FUNCTION_BLOCK COUNTER (* Composite Function Block Type *)
  (* Standard: 61499-2 *)
  (* Version 0.0, 2/4/2026, SESA713705, Schneider Electric, template *)
  PACKAGE SE.Nereda;
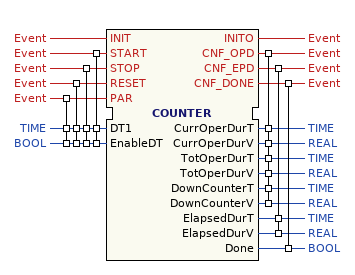
  EVENT_INPUT
    INIT;
    START WITH DT1, EnableDT; (* Begin Delay *)
    STOP WITH DT1, EnableDT; (* Cancel Delay *)
    RESET WITH DT1, EnableDT;
    PAR WITH DT1, EnableDT;
  END_EVENT
  EVENT_OUTPUT
    INITO;
    CNF_OPD WITH CurrOperDurT, CurrOperDurV, TotOperDurT, TotOperDurV, DownCounterT, DownCounterV; (* Execution Confirmation of current and total device operation duration *)
    CNF_EPD WITH ElapsedDurT, ElapsedDurV; (* Execution Confirmation of current and total Elapsed device duration *)
    CNF_DONE WITH Done;
  END_EVENT
  VAR_INPUT
    DT1 : TIME;
    EnableDT : BOOL;
  END_VAR
  VAR_OUTPUT
    CurrOperDurT : TIME;
    CurrOperDurV : REAL;
    TotOperDurT : TIME;
    TotOperDurV : REAL;
    DownCounterT : TIME;
    DownCounterV : REAL;
    ElapsedDurT : TIME;
    ElapsedDurV : REAL;
    Done : BOOL;
  END_VAR
  FBS
    IThis : COUNTER_HMI(QI := TRUE);
    CounterDurationCalc : devMntCalc(TBaseOperationDuration := T#1s, TBaseElapsedDuration := T#1d);
    CounterManager : CounterBasic;
    OPD : UDINT2TIME_2;
    REAL_OPD : UDINT2REAL_2;
    EPD_TIME : ElapsedTimeBasic;
    Counter : CounterSp;
    Smooth : boolValueChanged;
    DownCounteReal : SUB_2;
    Time2Real : TIME2REAL; {SET_ATTRIBUTE(Configuration.Component.HideUnusedPorts, )}
    Real2Time : REAL2TIME;
  END_FBS
  EVENT_CONNECTIONS
    CounterDurationCalc.INITO TO INITO;
    START TO CounterManager.DD7C28FB9184AAEE;
    STOP TO CounterManager.E0BAE2B19D215A1B;
    CounterManager.C2AFBA6527CC7C56 TO CounterDurationCalc.REQ_PV;
    Real2Time.79B40746AB555956 TO OPD.9954577AA24F9DD6;
    REAL_OPD.6FC99A5BD1C38561 TO CNF_OPD;
    EPD_TIME.B1E2A620E35E48BA TO CNF_EPD;
    OPD.79B40746AB555956 TO REAL_OPD.DD5870AA881150BB;
    REAL_OPD.6FC99A5BD1C38561 TO EPD_TIME.3E14346F747403ED;
    START TO EPD_TIME.90013566B02D29C0;
    STOP TO EPD_TIME.92EFFFA7C76F84E6;
    STOP TO EPD_TIME.3E14346F747403ED;
    Counter.C5DB08088DE67568 TO Smooth.REQ;
    PAR TO Counter.3BAEFB620E0425F5;
    REAL_OPD.6FC99A5BD1C38561 TO Counter.05FD3DED10D7909C;
    START TO Counter.C8BF0B5DBAF12ADE;
    STOP TO Counter.A678C75868BE7A7E;
    Smooth.CHD TO CNF_DONE;
    CounterDurationCalc.CNF_OPD TO Time2Real.9954577AA24F9DD6;
    PAR TO Time2Real.9954577AA24F9DD6;
    Time2Real.79B40746AB555956 TO DownCounteReal.DD5870AA881150BB;
    DownCounteReal.6FC99A5BD1C38561 TO Real2Time.9954577AA24F9DD6;
    INIT TO IThis.BDCD7F4C509A4BB9;
    REAL_OPD.6FC99A5BD1C38561 TO IThis.74F88D2B8EA734B3;
    EPD_TIME.B1E2A620E35E48BA TO IThis.CFA317C2D974F51D;
    PAR TO IThis.9D68FA4A40F281E7;
    REAL_OPD.6FC99A5BD1C38561 TO IThis.9D68FA4A40F281E7;
    IThis.17583D3249A041B7 TO CounterDurationCalc.INIT;
    RESET TO CounterManager.24B9D0C79B9A3EE2;
  END_CONNECTIONS
  DATA_CONNECTIONS
    CounterManager.C5D705445004F6D1 TO CounterDurationCalc.Pv;
    CounterDurationCalc.CurrentOperationDuration TO OPD.158B8AA7B31D2617;
    CounterDurationCalc.TotalOperationDuration TO OPD.E55D6D2AC87EFFD0;
    CounterDurationCalc.CurrentOperationDuration TO REAL_OPD.4573FC8F228EB71D;
    CounterDurationCalc.TotalOperationDuration TO REAL_OPD.63EF56506AEB9BC9;
    OPD.8AC404843F53B283 TO CurrOperDurT;
    OPD.4CB3A5FE1D5BD476 TO TotOperDurT;
    REAL_OPD.A6DEF5F9C27C1848 TO CurrOperDurV;
    REAL_OPD.5DAA0892996D1670 TO TotOperDurV;
    EPD_TIME.A1F07991DD7F26F4 TO ElapsedDurT;
    OPD.8AC404843F53B283 TO EPD_TIME.59105EE79BB5FB0A;
    EPD_TIME.CABA7EC1FA43F708 TO ElapsedDurV;
    CounterDurationCalc.CurrentOperationDuration TO EPD_TIME.C5E465A1E0BF9BC5;
    Counter.58C9703823A8F8AF TO Smooth.Input;
    DT1 TO Counter.2757200F630CD003;
    OPD.8AC404843F53B283 TO Counter.86924FE0C1577BC6;
    EnableDT TO Counter.CB3CEBB9E250D30E;
    Smooth.Output TO Done;
    DT1 TO Time2Real.158B8AA7B31D2617;
    Time2Real.8AC404843F53B283 TO DownCounteReal.4573FC8F228EB71D;
    REAL_OPD.A6DEF5F9C27C1848 TO DownCounteReal.ED82F6F6A6E0B1CD;
    DownCounteReal.A6DEF5F9C27C1848 TO Real2Time.158B8AA7B31D2617;
    Real2Time.8AC404843F53B283 TO DownCounterT;
    DownCounteReal.A6DEF5F9C27C1848 TO DownCounterV;
    OPD.8AC404843F53B283 TO IThis.7197075EDDE66C4;
    OPD.4CB3A5FE1D5BD476 TO IThis.A99CC2BF2705E5E2;
    EPD_TIME.A1F07991DD7F26F4 TO IThis.801397074C3CB402;
    DT1 TO IThis.BDE037A3D35B58AC;
    OPD.8AC404843F53B283 TO IThis.32801FF6D4B0F131;
    Real2Time.8AC404843F53B283 TO IThis.DD6B8E71CF375E06;
    CounterManager.DAD2EDD22719CB1D TO CounterDurationCalc.ResetOperationDuration;
  END_CONNECTIONS
END_FUNCTION_BLOCK
